FUNCTION_BLOCK FB_RotaryEncoder EXTENDS FB_HMIBase
VAR_INPUT
END_VAR
VAR_OUTPUT
END_VAR
VAR
END_VAR

END_FUNCTION_BLOCK

(* stored: Version 1.1.0.1
   POU FB_RotaryEncoder: Id {b03b6cc7-f3f4-4091-99dd-be277cfee204}, SpecialFunc None *)
